(* IEC 61131-3 sources: plc_generation_empirical_study/datasets/task_bank_c04_reverse_runtime_v0_3/tasks/C04_S05_lean_composite, 2 files *)

(* ---- interface.st ---- *)
FUNCTION_BLOCK C04_S05_lean_composite
VAR_INPUT
    A_Info : BOOL;
    A_Warning : BOOL;
    A_Trip : BOOL;
    A_Emergency : BOOL;
    A_Suppress : BOOL;
    B_EventA : BOOL;
    B_EventB : BOOL;
    B_Qualify : BOOL;
    B_Inhibit : BOOL;
    B_Reset : BOOL;
    B_MaxCount : INT;
    SubsystemBEnable : BOOL;
    CrossReset : BOOL;
END_VAR
VAR_OUTPUT
    A_Active : BOOL;
    A_Level : INT;
    B_PulseA : BOOL;
    B_PulseB : BOOL;
    B_Count : INT;
    B_Locked : BOOL;
    B_LastSource : INT;
    CrossReady : BOOL;
    CrossBlocked : BOOL;
END_VAR
END_FUNCTION_BLOCK

(* ---- reference.st ---- *)
FUNCTION_BLOCK C04_S05_lean_composite
VAR_INPUT
    A_Info : BOOL;
    A_Warning : BOOL;
    A_Trip : BOOL;
    A_Emergency : BOOL;
    A_Suppress : BOOL;
    B_EventA : BOOL;
    B_EventB : BOOL;
    B_Qualify : BOOL;
    B_Inhibit : BOOL;
    B_Reset : BOOL;
    B_MaxCount : INT;
    SubsystemBEnable : BOOL;
    CrossReset : BOOL;
END_VAR
VAR_OUTPUT
    A_Active : BOOL;
    A_Level : INT;
    B_PulseA : BOOL;
    B_PulseB : BOOL;
    B_Count : INT;
    B_Locked : BOOL;
    B_LastSource : INT;
    CrossReady : BOOL;
    CrossBlocked : BOOL;
END_VAR
VAR
    B_PrevA : BOOL;
    B_PrevB : BOOL;
END_VAR

IF A_Emergency THEN
    A_Level := 4;
    A_Active := TRUE;
ELSIF A_Suppress THEN
    A_Level := 0;
    A_Active := FALSE;
ELSIF A_Trip THEN
    A_Level := 3;
    A_Active := TRUE;
ELSIF A_Warning THEN
    A_Level := 2;
    A_Active := TRUE;
ELSIF A_Info THEN
    A_Level := 1;
    A_Active := TRUE;
ELSE
    A_Level := 0;
    A_Active := FALSE;
END_IF;

IF CrossReset THEN
    CrossReady := FALSE;
ELSIF A_Active THEN
    CrossReady := TRUE;
END_IF;
CrossBlocked := SubsystemBEnable AND (NOT CrossReady);

IF SubsystemBEnable AND CrossReady THEN
    B_PulseA := FALSE;
    B_PulseB := FALSE;
    IF B_Reset AND (NOT B_EventA) AND (NOT B_EventB) THEN
        B_Count := 0;
        B_Locked := FALSE;
        B_LastSource := 0;
    ELSIF B_MaxCount <= 0 THEN
        B_Locked := TRUE;
    ELSIF B_Qualify AND (NOT B_Inhibit) AND (NOT B_Locked) THEN
        IF B_EventA AND (NOT B_PrevA) THEN
            B_PulseA := TRUE;
            B_Count := B_Count + 1;
            B_LastSource := 1;
        ELSIF B_EventB AND (NOT B_PrevB) THEN
            B_PulseB := TRUE;
            B_Count := B_Count + 1;
            B_LastSource := 2;
        END_IF;
        IF B_Count >= B_MaxCount THEN B_Count := B_MaxCount; B_Locked := TRUE; END_IF;
    END_IF;
    B_PrevA := B_EventA;
    B_PrevB := B_EventB;
ELSE
    B_PulseA := FALSE;
    B_PulseB := FALSE;
    B_Count := 0;
    B_Locked := FALSE;
    B_LastSource := 0;
END_IF;

END_FUNCTION_BLOCK
